FUNCTION_BLOCK FB_SavePersistentData
VAR_INPUT
END_VAR
VAR_OUTPUT
END_VAR
VAR
	
	instFbClkPrgWritePersistentData: CLK_PRG;
	instFbWritePersistentData: FB_WritePersistentData;
	savePersisteData: BOOL;
	cpuPowerFailDetected: BOOL;
	writePersistentDataBusy: BOOL;
	writePersistentDataErr: BOOL;
	instFBSUpsBapi: FB_S_UPS_CX9020_U900;
	
	writePersistentDataErrId :UDINT;
END_VAR

VAR PERSISTENT
		
	saveCounter: DINT;

END_VAR
VAR // added by the converter: edge detectors and wires of the graphical bodies
    _w1 : DINT;
END_VAR

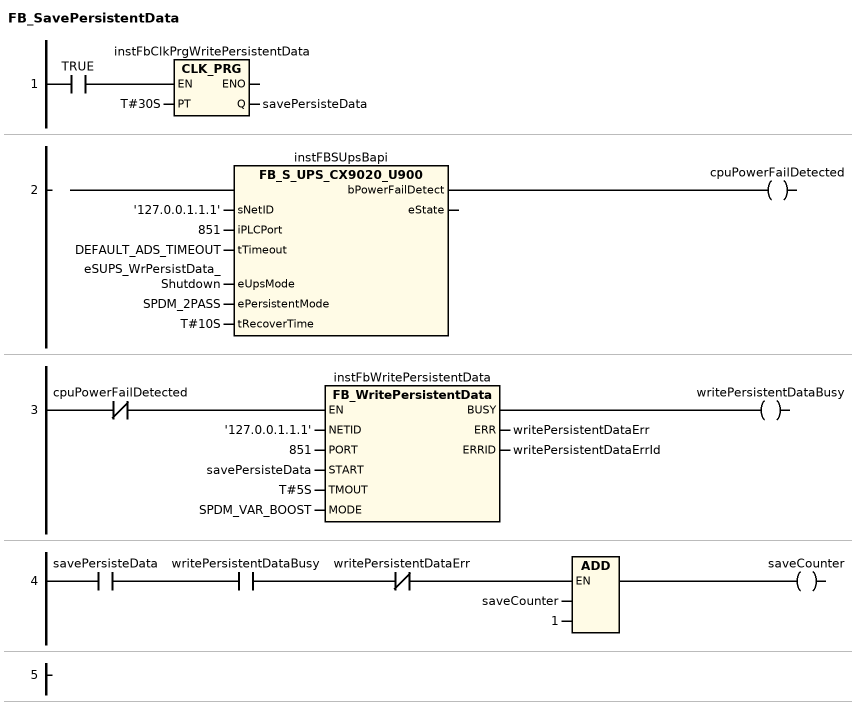
// NETWORK 1
instFbClkPrgWritePersistentData(PT := T#30S, Q => savePersisteData); // CLK_PRG

// NETWORK 2
instFBSUpsBapi(
    sNetID := '127.0.0.1.1.1',
    iPLCPort := 851,
    tTimeout := DEFAULT_ADS_TIMEOUT,
    eUpsMode := eSUPS_WrPersistData_Shutdown,
    ePersistentMode := SPDM_2PASS,
    tRecoverTime := T#10S); // FB_S_UPS_CX9020_U900
cpuPowerFailDetected := instFBSUpsBapi.bPowerFailDetect;

// NETWORK 3
IF NOT cpuPowerFailDetected THEN
    instFbWritePersistentData(
        NETID := '127.0.0.1.1.1',
        PORT := 851,
        START := savePersisteData,
        TMOUT := T#5S,
        MODE := SPDM_VAR_BOOST,
        ERR => writePersistentDataErr,
        ERRID => writePersistentDataErrId); // FB_WritePersistentData
END_IF
writePersistentDataBusy := instFbWritePersistentData.BUSY;

// NETWORK 4
IF savePersisteData AND writePersistentDataBusy AND NOT writePersistentDataErr THEN _w1 := saveCounter + 1; END_IF
saveCounter := _w1;

// NETWORK 5

END_FUNCTION_BLOCK

(* stored: Version 1.1.0.1
   POU FB_SavePersistentData: Id {c48c5cbd-c1fc-4744-a863-8aa8d68b6943}, SpecialFunc None *)
